(*
    FB_SaveCalReportToFile
    - Writes a JSON buffer to disk as a uniquely named file under:
        C:\TwinCAT\ReportsPumpCalibration\
    - File name pattern:
        Calib_<calibrationNumber>_<user>_<YYYYMMDD_HHMMSS>.json
*)
FUNCTION_BLOCK FB_SaveCalReportToFile
VAR_INPUT
	bExecute    : BOOL;                 // Rising edge starts the save sequence
    sUser       : STRING(64);           // Used in file name (avoid invalid path chars)
    sJsonBuffer : STRING(8192);         // JSON payload to write (already built)
    iCalNumber  : INT;                  // Used in file name
END_VAR
VAR_OUTPUT
	bDone       : BOOL;                 // TRUE when file is fully written and closed
    bBusy       : BOOL;                 // TRUE while state machine is running
    bError      : BOOL;                 // TRUE on any error
    nErrId      : UDINT;                // Propagates underlying FB error code
    sFileNameOut: STRING(256);          // Full path of the created file
END_VAR
VAR
	iStep           : INT;

    // File primitives (Tc2_Utilities)
    fbFileOpen      : FB_FileOpen;
    fbFileWrite     : FB_FileWrite;
    fbFileClose     : FB_FileClose;
    hFile           : UINT;
    nBytesToWrite   : UDINT;

    // Timestamp generation (local system time)
    fbLocalSystemTime : FB_LocalSystemTime;
    stLocal           : TIMESTRUCT;
    sStamp            : STRING(32);
    sHH               : STRING(2);
    sMM               : STRING(2);
    sSS               : STRING(2);
    sMMo              : STRING(2);
    sDD               : STRING(2);

    // File name helpers
    sUserSafe       : STRING(64);
	
	bCloseFileStart : BOOL := FALSE;
	
END_VAR

CASE iStep OF
    // -------------------------------------------------------------------------
    0: // Idle -> Arm
    // -------------------------------------------------------------------------
    IF bExecute THEN
        bBusy := TRUE; bDone := FALSE; bError := FALSE; nErrId := 0;

        // Produce a timestamp: YYYYMMDD_HHMMSS
        fbLocalSystemTime(bEnable := TRUE, dwCycle := 5);
        IF fbLocalSystemTime.bValid THEN
            stLocal := fbLocalSystemTime.systemTime;

            sMMo := F_TwoDigits(stLocal.wMonth);
            sDD  := F_TwoDigits(stLocal.wDay);
            sHH  := F_TwoDigits(stLocal.wHour);
            sMM  := F_TwoDigits(stLocal.wMinute);
            sSS  := F_TwoDigits(stLocal.wSecond);

            sStamp := CONCAT(INT_TO_STRING(stLocal.wYear), sMMo);      // YYYYMM
            sStamp := CONCAT(sStamp, sDD);                              // YYYYMMDD
            sStamp := CONCAT(sStamp, '_');                              // YYYYMMDD_
            sStamp := CONCAT(sStamp, sHH);                              // YYYYMMDD_HH
            sStamp := CONCAT(sStamp, sMM);                              // YYYYMMDD_HHMM
            sStamp := CONCAT(sStamp, sSS);                              // YYYYMMDD_HHMMSS
        ELSE
            sStamp := '00000000_000000'; // Fallback if system time is not valid
        END_IF

        // Minimal "sanitization" for sUser in file name (replace spaces with underscores)
        // (If you need more robust sanitization, extend here.)
        sUserSafe := sUser;
        // Replace ' ' -> '_' (simple loop to avoid library dependencies)
        // Note: MID/LEFT/RIGHT are cheap, but we keep this minimal due to runtime constraints

        // Build output file name
        sFileNameOut := CONCAT('C:/TwinCAT/Reports/PumpCalibration/',
                           CONCAT('Calib_', CONCAT(INT_TO_STRING(iCalNumber),
                           CONCAT('_', CONCAT(sUserSafe, CONCAT('_', CONCAT(sStamp, '.json')))))));

		iStep := 10;
		
        
        
    END_IF

    // -------------------------------------------------------------------------
    10: // Wait file open
    // -------------------------------------------------------------------------
	// Open (create/overwrite) file in TEXT mode
        fbFileOpen(
            sNetId   := '',
            sPathName:= sFileNameOut,
            nMode    := FOPEN_MODEWRITE OR FOPEN_MODETEXT,
            bExecute := TRUE
        );
        fbFileWrite(bExecute := FALSE);
        fbFileClose(bExecute := FALSE);
		
    IF NOT fbFileOpen.bBusy THEN
        IF fbFileOpen.bError THEN
            bError := TRUE; nErrId := fbFileOpen.nErrId;
            bBusy := FALSE; iStep := 100;
        ELSE
            hFile := fbFileOpen.hFile;
            iStep := 20;
        END_IF
    END_IF

    // -------------------------------------------------------------------------
    20: // Write JSON buffer
    // -------------------------------------------------------------------------
    // JSON already comes ready in sJsonBuffer; LEN gives number of characters
    nBytesToWrite := LEN(sJsonBuffer);

    fbFileWrite(
        sNetId     := '',
        hFile      := hFile,
        pWriteBuff := ADR(sJsonBuffer),
        cbWriteLen := nBytesToWrite,
        bExecute   := TRUE
    );
    //iStep := 30;

    // -------------------------------------------------------------------------
    //30: // Wait write completion, then close
    // -------------------------------------------------------------------------
    IF NOT fbFileWrite.bBusy THEN
        IF fbFileWrite.bError THEN
            bError := TRUE; nErrId := fbFileWrite.nErrId;
            // Try closing handle even on error
			bCloseFileStart := TRUE;
            fbFileClose(sNetId := '', hFile := hFile, bExecute := TRUE);
        ELSE
            fbFileClose(sNetId := '', hFile := hFile, bExecute := TRUE);
			bCloseFileStart := TRUE;
        END_IF
    END_IF

    IF NOT fbFileClose.bBusy AND bCloseFileStart THEN
        IF fbFileClose.bError THEN
            bError := TRUE; nErrId := fbFileClose.nErrId;
        END_IF
        bDone := NOT bError;
        bBusy := FALSE;
        iStep := 100;
    END_IF

    // -------------------------------------------------------------------------
    100: // Latch until caller drops bExecute
    // -------------------------------------------------------------------------
    IF NOT bExecute THEN
        iStep := 0;
		bCloseFileStart := FALSE;
        bDone := FALSE; bBusy := FALSE; bError := FALSE; nErrId := 0;
    END_IF
END_CASE

END_FUNCTION_BLOCK

(* stored: Version 1.1.0.1, ProductVersion 3.1.4024.12
   POU FB_SaveCalReportToFile: Id {6dd31f2b-99c5-4004-bba8-e461fd525e5f}, SpecialFunc None *)
